FUNCTION_BLOCK FutureMCGearOutCreator IMPLEMENTS I_TaskCreator
VAR_INPUT
END_VAR
VAR_OUTPUT
END_VAR
VAR
	_axis_sub: REFERENCE TO AXIS_REF;
	_option : ST_GearOutOptions;
END_VAR

{warning 'add method implementation '}
METHOD create_future : I_Future
VAR_INPUT
	(* Specify future name*)
	future_name	: STRING;
END_VAR
VAR
	_p_future : POINTER TO FutureMCGearOut;
END_VAR
_p_future := __NEW(FutureMCGearOut);
_p_future^.future_name := future_name;
_p_future^.set_parameters(_axis_sub);
_p_future^.set_options(_option);
create_future := _p_future^;
END_METHOD

{warning 'add method implementation '}
METHOD destroy_future : I_Future
VAR_INPUT
	(* Specify future instance whtat you want to delete.*)
	future	: I_Future;
END_VAR
VAR
	_p_future : POINTER TO FutureMCGearOut;
END_VAR
IF __QUERYPOINTER(future, _p_future) THEN
	__DELETE(_p_future);
	IF _p_future = 0  THEN
		destroy_future := 0;
	END_IF
END_IF
END_METHOD

METHOD set_options : BOOL
VAR_INPUT
	option : ST_GearOutOptions;
END_VAR
_option := option;
END_METHOD

METHOD set_parameters : BOOL
VAR_INPUT
	axis_sub : REFERENCE TO AXIS_REF;
END_VAR
_axis_sub REF= axis_sub;
END_METHOD

END_FUNCTION_BLOCK

(* stored: Version 1.1.0.1, ProductVersion 3.1.4026.17
   POU FutureMCGearOutCreator: Id {4f5e0dea-75bb-4c96-a76e-81abf884507a}, SpecialFunc None
   Method create_future: Id {475698ab-0737-47d6-8622-d026d33ab716}
   Method destroy_future: Id {8742e7d8-6813-4916-908a-50d4451908ac}
   Method set_options: Id {bee32503-b031-4440-a5fe-f846a91c0492}
   Method set_parameters: Id {7e618896-3ab5-45a7-82df-6c0f1a88332d} *)
